{attribute 'qualified_only'}
{attribute 'strict'}
{attribute 'to_string'}
// Log level of message to be logged.
TYPE E_LogLevel :
(
	Debug,
	Information,
	Warning,
	Error,
	Fatal
);
END_TYPE

(* stored: Version 1.1.0.1, ProductVersion 3.1.4024.4
   DUT E_LogLevel: Id {b22d3fef-91d4-49da-9c4a-eb3786bf2a9d} *)
